// TIA Portal V19 export
TYPE "lexchangetray_typeUnEmn_toHandlingXyzFeedback"
// Type: Bool
// stored: Access Published
   STRUCT
      catchEnable : Bool;   // 允许抓取
   END_STRUCT;
END_TYPE
